FUNCTION_BLOCK Station IMPLEMENTS IStation
VAR_INPUT
END_VAR
VAR_OUTPUT
END_VAR
VAR
	_Clear : BOOL;
	_Complete : BOOL;
	_Operating : BOOL;
	_Ready : BOOL;
	_Positions : ARRAY[1..4] OF MC_LREAL := [0.0,0.0,0.0,0.0];
	NumberOfPositions : INT := 0;
	AssignedPositions : INT := 1;
	StationMovers : INT;
	stInfo : stStationInfo;
	_HasMover : BOOL;
	ProductCounter : R_TRIG;
	Products : DINT;
	LastStation : BOOL;
	MyMover : IMover;
END_VAR

//Cyclic info
stInfo.StationPosition := _Positions[1];
stInfo.StationStatus.Clear := _clear;
stInfo.StationStatus.Complete := _Complete;
stInfo.StationStatus.HasMover := _HasMover;
stInfo.StationStatus.Operating := _Operating;
stInfo.StationStatus.Ready := _Ready;

IF LastStation THEN
	ProductCounter(CLK := _Complete);
	IF ProductCounter.Q THEN
		Products := Products + 1;
	END_IF
END_IF

METHOD Abort : BOOL
VAR_INPUT
END_VAR
_Complete := FALSE;
_Clear := TRUE;
_Operating := FALSE;
_Ready := TRUE;
END_METHOD

METHOD HasMover : BOOL
VAR_INPUT
	mover : IMover;
END_VAR
StationMovers := StationMovers + 1;
IF StationMovers = NumberOfPositions THEN
	_HasMover := TRUE;
END_IF
MyMover := mover;
END_METHOD

METHOD IsClear : BOOL
IsClear := _Clear;
END_METHOD

METHOD isComplete : BOOL
isComplete := _Complete;
END_METHOD

PROPERTY PUBLIC IsLastStation : BOOL
GET
IsLastStation := LastStation;
END_GET
SET
LastStation := IsLastStation;
END_SET
END_PROPERTY

METHOD IsOperating : BOOL
IsOperating := _Operating;
END_METHOD

METHOD IsReady : BOOL
IsReady := _Ready;
END_METHOD

METHOD MoverAway : BOOL
VAR_INPUT
END_VAR
StationMovers := StationMovers - 1;
MyMover := 0;
END_METHOD

PROPERTY Position : MC_LREAL
GET
Position := _Positions[AssignedPositions];
AssignedPositions := AssignedPositions + 1;
IF AssignedPositions > NumberOfPositions THEN
	AssignedPositions := 1;
END_IF
END_GET
SET
IF NumberOfPositions < 5 THEN
	NumberOfPositions := NumberOfPositions + 1;
	_Positions[NumberOfPositions] := Position;
END_IF
END_SET
END_PROPERTY

END_FUNCTION_BLOCK

(* stored: Version 1.1.0.1, ProductVersion 3.1.4024.12
   POU Station: Id {15da8106-0d22-4ca5-af9c-31c3d97b8668}, SpecialFunc None
   Method Abort: Id {38f6b9e4-2f32-4b37-b901-e23947342ba9}
   Method HasMover: Id {1cb719ab-8b5a-456f-a91b-48331f9d0dc2}
   Method IsClear: Id {76a4496f-67c0-45fc-9e15-a528954fd797}
   Method isComplete: Id {e952f541-8c98-4290-8bef-72b636ded12c}
   Property IsLastStation: Id {a73398cf-8042-40d8-a8fb-0a856e7df54f}
   Get Get: Id {9cd8ec45-e245-4fd5-a342-74a5c351fecb}
   Set Set: Id {71583b8e-176c-4a77-8f64-6a07e8be2663}
   Method IsOperating: Id {46f6a6eb-2d48-45d2-a61c-982a5af29ec7}
   Method IsReady: Id {72424547-540c-4f0b-8c61-f3533ca0048c}
   Method MoverAway: Id {5bac361c-272f-42b5-96ba-9a558f55b3c0}
   Property Position: Id {4a10e32c-305e-441b-9332-8642baafa7cc}
   Get Get: Id {6760ec00-0cdd-4667-9f90-fd015738ea5e}
   Set Set: Id {825e159a-d125-4194-a2b1-af8249a79ce1} *)
